// TIA Portal V17 export
// export: Created 2024-09-02T12:50:08.1764896Z, ExportSetting WithDefaults, DisplayName Totally Integrated Automation Portal, DisplayVersion V17, DisplayName TIA Portal Openness, DisplayVersion V17, DisplayName TIA Portal Version Control Interface, DisplayVersion V17, DisplayName STEP 7 Professional, DisplayVersion V17, DisplayName STEP 7 Safety, DisplayVersion V17, DisplayName WinCC Professional, DisplayVersion V17
FUNCTION_BLOCK "GraFB9_FG02_Home_OP70"   // FB1389, GRAPH
VERSION : 0.1
// stored: AcknowledgeErrorsRequired true, AutoNumber false, GraphVersion 4.0, InitialValuesAcquisition false, IsIECCheckEnabled false, LanguageInNetworks LAD, LockOperatingMode false, PermanentILProcessingInMANMode true, SetENOAutomatically false, SkipSteps false, UDAEnableTagReadback false, WithAlarmHandling true
   // inherited from GRAPH_BASE
   VAR
      OFF_SQ_BASE : Bool;
   END_VAR
   VAR_INPUT
      OFF_SQ { ExternalWritable := 'False'} : Bool := false;   // Kette ausschalten / Turn sequence off
      INIT_SQ { ExternalWritable := 'False'} : Bool := false;   // Kette in Initialzustand versetzen / Set sequence to initial state
      ACK_EF { ExternalWritable := 'False'} : Bool := false;   // Alle Fehler und Störungen quittieren / Acknowledge all errors and faults
      S_PREV { ExternalWritable := 'False'} : Bool := false;   // Vorherigen Schritt am Parameter S_NO ausgeben / Output previous step in parameter S_NO
      S_NEXT { ExternalWritable := 'False'} : Bool := false;   // Nächsten Schritt am Parameter S_NO anzeigen / Indicate next step in parameter S_NO
      SW_AUTO { ExternalWritable := 'False'} : Bool := false;   // Automtischer Betrieb / Automatic mode
      SW_TAP { ExternalWritable := 'False'} : Bool := false;   // Halbautomatisch/Weiterschalten mit Transition / Semiautomatic/switch with transition
      SW_TOP { ExternalWritable := 'False'} : Bool := false;   // Halbautomatisch/Ignoriere Transition / Semiautomatic/ignore transition
      SW_MAN { ExternalWritable := 'False'} : Bool := false;   // Handbetrieb / Manual mode
      S_SEL { ExternalWritable := 'False'} : Int := 0;   // Schritt auswählen, der an S_NO ausgegeben werden soll / Select step to be output to S_NO
      S_ON { ExternalWritable := 'False'} : Bool := false;   // Schritt aktivieren, der an Parameter S_NO anliegt / Activate step indicated in S_NO
      S_OFF { ExternalWritable := 'False'} : Bool := false;   // Schritt deaktivieren, der an Parameter S_NO anliegt / Deactivate step indicated S_NO
      T_PUSH { ExternalWritable := 'False'} : Bool := false;   // Schaltfreigabe für Transition im halbautomatischen Betrieb / Enable transition to switch in semi automatic mode
   END_VAR
   VAR_OUTPUT
      S_NO { ExternalWritable := 'False'} : Int := 0;   // Schrittnummer / Step number
      S_MORE { ExternalWritable := 'False'} : Bool := false;   // Weitere Schritte sind vorhanden und können in S_NO angezeigt werden. / More steps are available and can be shown in S_NO
      S_ACTIVE { ExternalWritable := 'False'} : Bool := false;   // Schritt, der an Parameter S_NO angezeigt wird, ist aktiv / Step indicated in S_NO is active
      ERR_FLT { ExternalWritable := 'False'} : Bool := false;   // Sammelfehler Interlock oder Supervision / Interlock or supervision group error
      AUTO_ON { ExternalWritable := 'False'} : Bool := false;   // Automatischer Betrieb eingeschaltet / Automatic mode is active
      TAP_ON { ExternalWritable := 'False'} : Bool := false;   // Halbautomatischer Betrieb/Schritt mit Transition eingeschaltet / Semiautomatic mode/step with transition enabled
      TOP_ON { ExternalWritable := 'False'} : Bool := false;   // Halbautomatischer Betrieb/Ignoriere Transition eingeschaltet / Semiautomatic mode/ignore transition enabled
      MAN_ON { ExternalWritable := 'False'} : Bool := false;   // Handbetrieb eingeschaltet / Manual mode is active
   END_VAR
   VAR
      extBlock { S7_SetPoint := 'True'} : "LTLL_ManualGraphExt";
   END_VAR
BEGIN
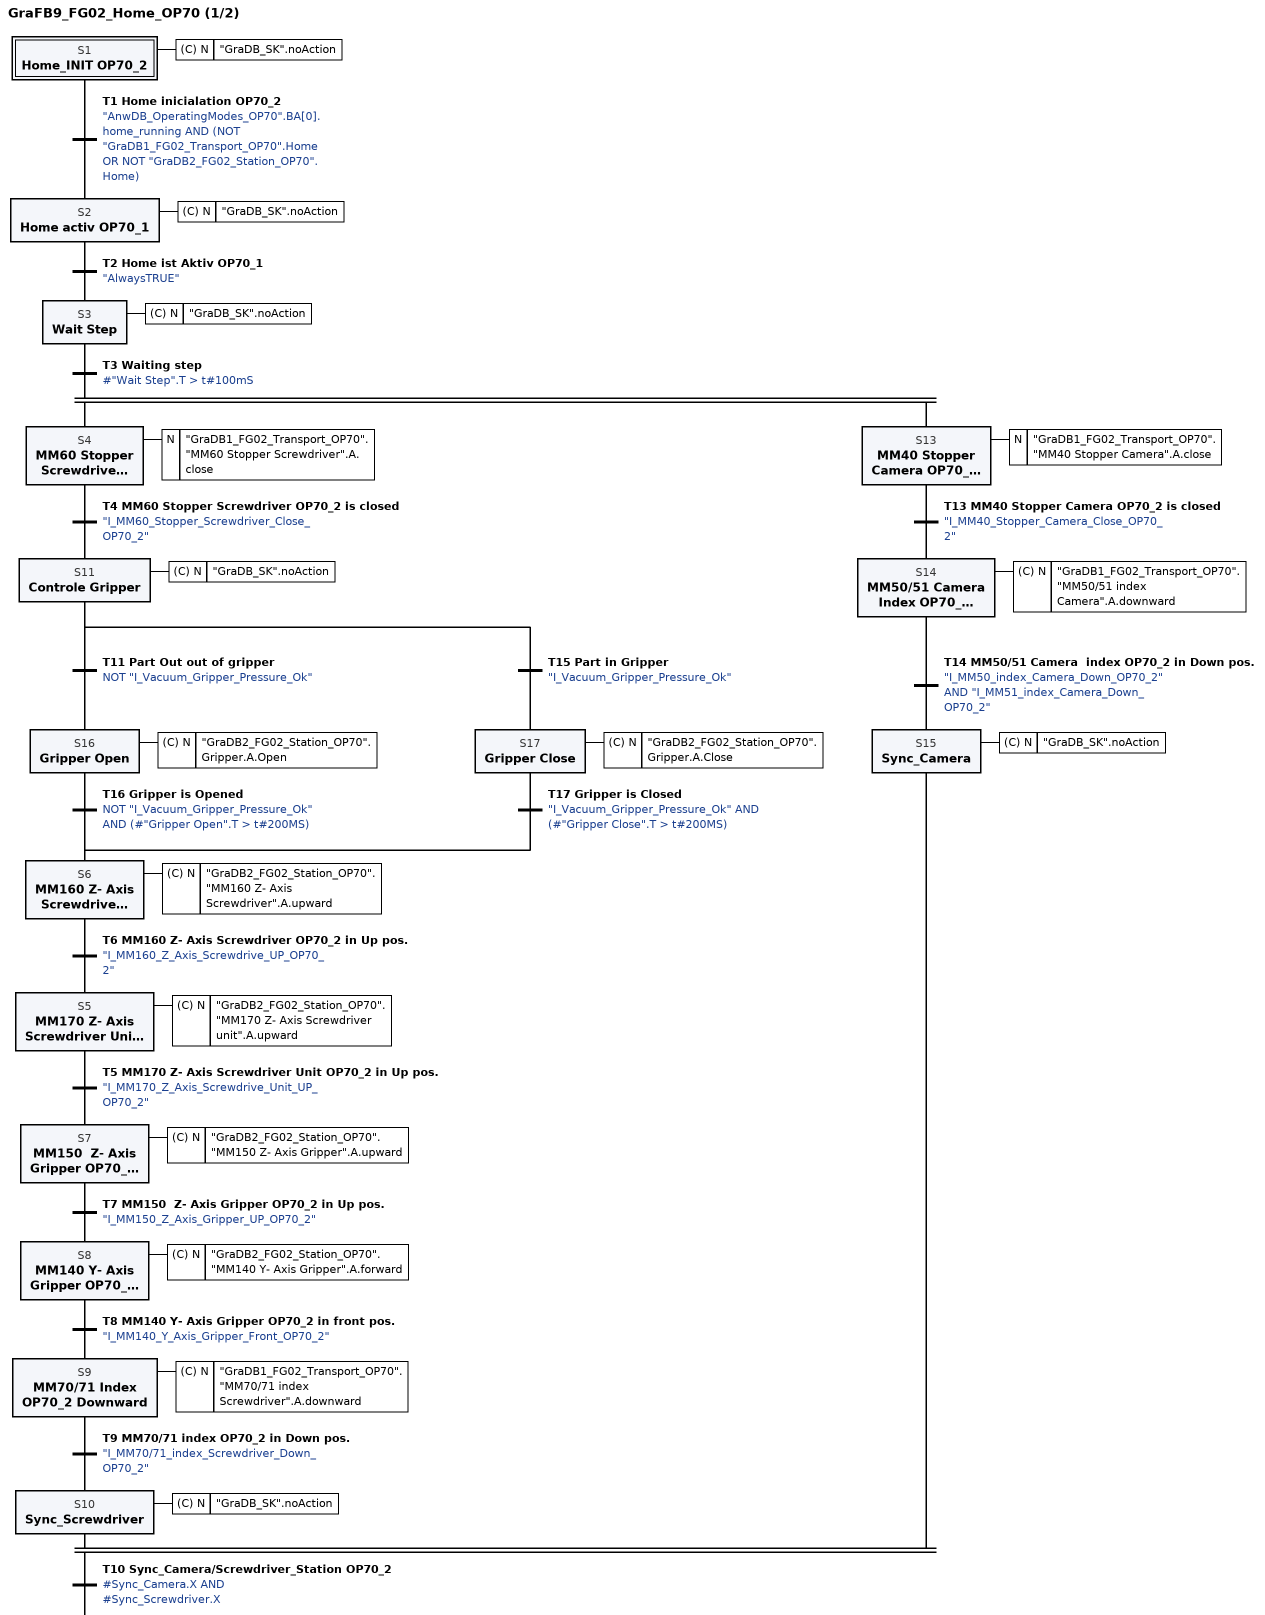
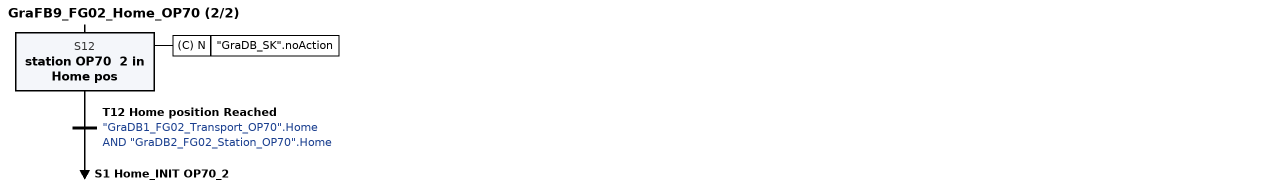
   // permanent pre-instructions
   NETWORK 1
   TITLE = HMI Lite Pass on data / HMI Lite Daten weiterreichen
      #extBlock.input := "LTLL_ManualGraphControl_OP70".screen[0].input;
   NETWORK 2
   TITLE = Instance DB Name query and pass on / Instanz DB Name abfragen und weiterreichen
      GetInstanceName(size := 0, OUT => #extBlock.input.instanceName);
   NETWORK 3
   TITLE = SK Mode
      "SysFC_SQ_Mode"(iFKT := 0, iTmsHalt := false, ioMOP := #RT_DATA.MOP);

   // sequencer 1: basic position drive / Grundstellungsfahrt
   INITIAL_STEP "Home_INIT OP70_2":   // S1, max time T#10S, warning time T#7S: Step commentary / Schrittkommentar
      interlock C := (none);   // Initialschritt / initial step
      supervision V := (none);   // Initialschritt / initial step
      (C)     N    "GraDB_SK".noAction
   END_STEP
   TRANSITION "Home inicialation OP70_2" FROM "Home_INIT OP70_2" TO "Home activ OP70_1"   // T1
      := "AnwDB_OperatingModes_OP70".BA[0].home_running AND (NOT "GraDB1_FG02_Transport_OP70".Home OR NOT "GraDB2_FG02_Station_OP70".Home);
   END_TRANSITION
   STEP "Home activ OP70_1":   // S2, max time T#10S, warning time T#7S
      supervision V := NOT #"Home ist Aktiv OP70_1".TT AND (#"Home activ OP70_1".U > T#5S);
      (C)     N    "GraDB_SK".noAction
   END_STEP
   TRANSITION "Home ist Aktiv OP70_1" FROM "Home activ OP70_1" TO "Wait Step"   // T2
      := "AlwaysTRUE";
   END_TRANSITION
   STEP Sync_Screwdriver:   // S10, max time T#10S, warning time T#7S: Step commentary / Schrittkommentar
      interlock C := (none);   // Initialschritt / initial step
      supervision V := (none);   // Initialschritt / initial step
      (C)     N    "GraDB_SK".noAction
   END_STEP
   TRANSITION "Sync_Camera/Screwdriver_Station OP70_2" FROM (Sync_Camera, Sync_Screwdriver) TO "station OP70  2 in Home pos"   // T10
      := #Sync_Camera.X AND #Sync_Screwdriver.X;
   END_TRANSITION
   STEP "MM150  Z- Axis Gripper OP70_2 Upward":   // S7, max time T#10S, warning time T#7S
      interlock C := "I_MM160_Z_Axis_Screwdrive_UP_OP70_2" AND "I_MM170_Z_Axis_Screwdrive_Unit_UP_OP70_2" AND (NOT "AnwDB_ProcessData_FG02_OP70".BEA[3].Complete.OK OR ("AnwDB_ProcessData_FG02_OP70".BEA[3].Complete.OK AND NOT "I_Vacuum_Gripper_Pressure_Ok"));
      supervision V := NOT #"MM150  Z- Axis Gripper OP70_2 in Up pos.".TT AND (#"MM150  Z- Axis Gripper OP70_2 Upward".U > T#5S);
      (C)     N    "GraDB2_FG02_Station_OP70"."MM150 Z- Axis Gripper".A.upward
   END_STEP
   TRANSITION "MM150  Z- Axis Gripper OP70_2 in Up pos." FROM "MM150  Z- Axis Gripper OP70_2 Upward" TO "MM140 Y- Axis Gripper OP70_2 Forward"   // T7
      := "I_MM150_Z_Axis_Gripper_UP_OP70_2";
   END_TRANSITION
   STEP "MM60 Stopper Screwdriver OP70_2 Closing":   // S4, max time T#10S, warning time T#7S
      supervision V := NOT #"MM60 Stopper Screwdriver OP70_2 is closed".TT AND (#"MM60 Stopper Screwdriver OP70_2 Closing".U > T#5S);
              N    "GraDB1_FG02_Transport_OP70"."MM60 Stopper Screwdriver".A.close
   END_STEP
   TRANSITION "MM60 Stopper Screwdriver OP70_2 is closed" FROM "MM60 Stopper Screwdriver OP70_2 Closing" TO "Controle Gripper"   // T4
      := "I_MM60_Stopper_Screwdriver_Close_OP70_2";
   END_TRANSITION
   STEP "MM40 Stopper Camera OP70_2 Closing":   // S13, max time T#10S, warning time T#7S
      supervision V := NOT #"MM40 Stopper Camera OP70_2 is closed".TT AND (#"MM40 Stopper Camera OP70_2 Closing".U > T#5S);
              N    "GraDB1_FG02_Transport_OP70"."MM40 Stopper Camera".A.close
   END_STEP
   TRANSITION "MM40 Stopper Camera OP70_2 is closed" FROM "MM40 Stopper Camera OP70_2 Closing" TO "MM50/51 Camera Index OP70_2 Downward"   // T13
      := "I_MM40_Stopper_Camera_Close_OP70_2";
   END_TRANSITION
   STEP "MM160 Z- Axis Screwdriver OP70_2 Upward":   // S6, max time T#10S, warning time T#7S
      interlock C := "AlwaysTRUE";
      supervision V := NOT #"MM160 Z- Axis Screwdriver OP70_2 in Up pos.".TT AND (#"MM160 Z- Axis Screwdriver OP70_2 Upward".U > T#5S);
      (C)     N    "GraDB2_FG02_Station_OP70"."MM160 Z- Axis Screwdriver".A.upward
   END_STEP
   TRANSITION "MM160 Z- Axis Screwdriver OP70_2 in Up pos." FROM "MM160 Z- Axis Screwdriver OP70_2 Upward" TO "MM170 Z- Axis Screwdriver Unit OP70_2 Upward"   // T6
      := "I_MM160_Z_Axis_Screwdrive_UP_OP70_2";
   END_TRANSITION
   STEP "MM50/51 Camera Index OP70_2 Downward":   // S14, max time T#10S, warning time T#7S
      interlock C := "AlwaysTRUE";
      supervision V := NOT #"MM50/51 Camera  index OP70_2 in Down pos.".TT AND (#"MM50/51 Camera Index OP70_2 Downward".U > T#5S);
      (C)     N    "GraDB1_FG02_Transport_OP70"."MM50/51 index Camera".A.downward
   END_STEP
   TRANSITION "MM50/51 Camera  index OP70_2 in Down pos." FROM "MM50/51 Camera Index OP70_2 Downward" TO Sync_Camera   // T14
      := "I_MM50_index_Camera_Down_OP70_2" AND "I_MM51_index_Camera_Down_OP70_2";
   END_TRANSITION
   STEP Sync_Camera:   // S15, max time T#10S, warning time T#7S: Step commentary / Schrittkommentar
      interlock C := (none);   // Initialschritt / initial step
      supervision V := (none);   // Initialschritt / initial step
      (C)     N    "GraDB_SK".noAction
   END_STEP
   STEP "MM140 Y- Axis Gripper OP70_2 Forward":   // S8, max time T#10S, warning time T#7S
      interlock C := "I_MM150_Z_Axis_Gripper_UP_OP70_2" AND "I_MM160_Z_Axis_Screwdrive_UP_OP70_2" AND "I_MM170_Z_Axis_Screwdrive_Unit_UP_OP70_2";
      supervision V := NOT #"MM140 Y- Axis Gripper OP70_2 in front pos.".TT AND (#"MM140 Y- Axis Gripper OP70_2 Forward".U > T#5S);
      (C)     N    "GraDB2_FG02_Station_OP70"."MM140 Y- Axis Gripper".A.forward
   END_STEP
   TRANSITION "MM140 Y- Axis Gripper OP70_2 in front pos." FROM "MM140 Y- Axis Gripper OP70_2 Forward" TO "MM70/71 Index OP70_2 Downward"   // T8
      := "I_MM140_Y_Axis_Gripper_Front_OP70_2";
   END_TRANSITION
   STEP "MM70/71 Index OP70_2 Downward":   // S9, max time T#10S, warning time T#7S
      interlock C := "I_MM150_Z_Axis_Gripper_UP_OP70_2" AND "I_MM160_Z_Axis_Screwdrive_UP_OP70_2" AND "I_MM170_Z_Axis_Screwdrive_Unit_UP_OP70_2";
      supervision V := NOT #"MM70/71 index OP70_2 in Down pos.".TT AND (#"MM70/71 Index OP70_2 Downward".U > T#5S);
      (C)     N    "GraDB1_FG02_Transport_OP70"."MM70/71 index Screwdriver".A.downward
   END_STEP
   TRANSITION "MM70/71 index OP70_2 in Down pos." FROM "MM70/71 Index OP70_2 Downward" TO Sync_Screwdriver   // T9
      := "I_MM70/71_index_Screwdriver_Down_OP70_2";
   END_TRANSITION
   STEP "MM170 Z- Axis Screwdriver Unit OP70_2 Upward":   // S5, max time T#10S, warning time T#7S
      interlock C := "I_Safety_bolt_Z_Axis_Screwdrive";
      supervision V := NOT #"MM170 Z- Axis Screwdriver Unit OP70_2 in Up pos.".TT AND (#"MM170 Z- Axis Screwdriver Unit OP70_2 Upward".U > T#5S);
      (C)     N    "GraDB2_FG02_Station_OP70"."MM170 Z- Axis Screwdriver unit".A.upward
   END_STEP
   TRANSITION "MM170 Z- Axis Screwdriver Unit OP70_2 in Up pos." FROM "MM170 Z- Axis Screwdriver Unit OP70_2 Upward" TO "MM150  Z- Axis Gripper OP70_2 Upward"   // T5
      := "I_MM170_Z_Axis_Screwdrive_Unit_UP_OP70_2";
   END_TRANSITION
   STEP "Wait Step":   // S3, max time T#10S, warning time T#7S
      supervision V := NOT #"Waiting step".TT AND (#"Wait Step".U > T#5S);
      (C)     N    "GraDB_SK".noAction
   END_STEP
   TRANSITION "Waiting step" FROM "Wait Step" TO ("MM60 Stopper Screwdriver OP70_2 Closing", "MM40 Stopper Camera OP70_2 Closing")   // T3
      := #"Wait Step".T > t#100mS;
   END_TRANSITION
   STEP "station OP70  2 in Home pos":   // S12, max time T#10S, warning time T#7S
      (C)     N    "GraDB_SK".noAction
   END_STEP
   TRANSITION "Home position Reached" FROM "station OP70  2 in Home pos" TO "Home_INIT OP70_2"   // T12, jump
      := "GraDB1_FG02_Transport_OP70".Home AND "GraDB2_FG02_Station_OP70".Home;
   END_TRANSITION
   STEP "Controle Gripper":   // S11, max time T#10S, warning time T#7S
      supervision V := NOT #"Part Out out of gripper".TT AND (#"Controle Gripper".U > T#5S);
      (C)     N    "GraDB_SK".noAction
   END_STEP
   TRANSITION "Part Out out of gripper" FROM "Controle Gripper" TO "Gripper Open"   // T11
      := NOT "I_Vacuum_Gripper_Pressure_Ok";
   END_TRANSITION
   TRANSITION "Part in Gripper" FROM "Controle Gripper" TO "Gripper Close"   // T15
      := "I_Vacuum_Gripper_Pressure_Ok";
   END_TRANSITION
   STEP "Gripper Open":   // S16, max time T#10S, warning time T#7S
      interlock C := "AlwaysTRUE";
      supervision V := NOT #"Gripper is Opened".TT AND (#"Gripper Open".U > T#5S);
      (C)     N    "GraDB2_FG02_Station_OP70".Gripper.A.Open
   END_STEP
   TRANSITION "Gripper is Opened" FROM "Gripper Open" TO "MM160 Z- Axis Screwdriver OP70_2 Upward"   // T16
      := NOT "I_Vacuum_Gripper_Pressure_Ok" AND (#"Gripper Open".T > t#200MS);
   END_TRANSITION
   STEP "Gripper Close":   // S17, max time T#10S, warning time T#7S
      interlock C := "AlwaysTRUE";
      supervision V := NOT #"Gripper is Closed".TT AND (#"Gripper Close".U > T#5S);
      (C)     N    "GraDB2_FG02_Station_OP70".Gripper.A.Close
   END_STEP
   TRANSITION "Gripper is Closed" FROM "Gripper Close" TO "MM160 Z- Axis Screwdriver OP70_2 Upward"   // T17
      := "I_Vacuum_Gripper_Pressure_Ok" AND (#"Gripper Close".T > t#200MS);
   END_TRANSITION

   // permanent post-instructions
   NETWORK 1
   TITLE = Move interlocks from Ext block to ManualGraphControl DB / Interlocks vom Ext-Block zum ManualGraphControl DB rangieren
      "LTLL_ManualGraphInterlock"(ManualGraphExtOutput := #extBlock.output,
                              ManualGraphControlScreen := "LTLL_ManualGraphControl_OP70".screen[0]);
   NETWORK 2
   TITLE = Report step error / Schrittkettenfehler melden
      "SysFC_NumOfSQErrors"(FLT := #RT_DATA.SQ_FLAGS.ERR_FLT,
                            Fault_SQ := "AnwDB_OperatingModes_OP70".BA[0].error_report_SK,
                            NumOf_Fault_SQ := "AnwDB_ZP_Alarm_OP70".FaultsNoSK_ST1);
   NETWORK 3
   TITLE = SK in home position / SK in Grundstellung
      "GraDB_Home".OP70_2.Home_SK := #"Home_INIT OP70_2".X;
END_FUNCTION_BLOCK
